// TwinCAT 3 PLC project Sample01
// ProgramVersion: 3.1.4023.0
// libraries:
//   Tc2_Standard, * (Beckhoff Automation GmbH)
//   Tc2_System, * (Beckhoff Automation GmbH)
//   Tc3_Module, * (Beckhoff Automation GmbH)
// project tree:
//   DUTs/ E_SortedOrder.TcDUT, ST_SequenceItem.TcDUT
//   / PlcTask.TcTTO
//   POUs/ Class Diagram.TcCD (not stored), FB_SequenceManager.TcPOU, MAIN.TcPOU
// real-time tasks:
//   TASK PlcTask: cycle T#10ms, priority 20, ADS port 350

CONFIGURATION Sample01
    RESOURCE PLC ON TwinCAT3
        TASK PlcTask(INTERVAL := T#10ms, PRIORITY := 20);
        PROGRAM MAIN WITH PlcTask : MAIN;
    END_RESOURCE
END_CONFIGURATION

// ---- DUTs/E_SortedOrder.TcDUT
{attribute 'qualified_only'}
{attribute 'strict'}
TYPE E_SortedOrder :
(
	Id,
	Value
);
END_TYPE

// ---- DUTs/ST_SequenceItem.TcDUT
TYPE ST_SequenceItem :
STRUCT
	nId			: UINT;
	nValue		: USINT(0..100);
	nDuration	: UINT; 
END_STRUCT
END_TYPE

// ---- POUs/MAIN.TcPOU
PROGRAM MAIN
VAR
	fbPlayList		: FB_SequenceManager;
	nTest			: INT;
END_VAR

IF (nTest = 1) THEN
	fbPlayList.Sort(E_SortedOrder.Id);
	nTest := 0;
ELSIF (nTest = 2) THEN
	fbPlayList.Sort(E_SortedOrder.Value);
	nTest := 0;
END_IF

END_PROGRAM

// ---- POUs/FB_SequenceManager.TcPOU
FUNCTION_BLOCK PUBLIC FB_SequenceManager
VAR_INPUT
END_VAR
VAR_OUTPUT
END_VAR
VAR
	// backing variable
	_aSequence	: ARRAY [1..5] OF ST_SequenceItem := [(nId := 1, nValue := 50, nDuration := 20),
													  (nId := 2, nValue := 10, nDuration := 30),
													  (nId := 3, nValue := 23, nDuration := 10),
													  (nId := 4, nValue := 65, nDuration := 200),
													  (nId := 5, nValue := 45, nDuration := 75)];
END_VAR

{attribute 'monitoring' := 'variable'}
PROPERTY PUBLIC aSequence : ARRAY [1..5] OF ST_SequenceItem
GET
aSequence := _aSequence;
END_GET
SET // PROTECTED
_aSequence := aSequence;
END_SET
END_PROPERTY

METHOD PUBLIC Sort
VAR_INPUT
	eSortedOrder		: E_SortedOrder;
END_VAR
VAR
	stLeft, stRight		: ST_SequenceItem;
	nMax, nIndex		: DINT;
	bSwapped			: BOOL;
END_VAR
CASE eSortedOrder OF
	E_SortedOrder.Id:
		REPEAT
			bSwapped := FALSE;
			FOR nIndex := 1 TO 4 DO
				stLeft := THIS^._aSequence[nIndex];
				stRight := THIS^._aSequence[nIndex + 1];
				IF (stLeft.nId > stRight.nId) THEN
					THIS^._aSequence[nIndex + 1] := stLeft;
					THIS^._aSequence[nIndex] := stRight;
					bSwapped := TRUE;
				END_IF
			END_FOR
		UNTIL
			bSwapped = FALSE
		END_REPEAT;

	E_SortedOrder.Value:
		REPEAT
			bSwapped := FALSE;
			FOR nIndex := 1 TO 4 DO
				stLeft := THIS^._aSequence[nIndex];
				stRight := THIS^._aSequence[nIndex + 1];
				IF (stLeft.nValue > stRight.nValue) THEN
					THIS^._aSequence[nIndex + 1] := stLeft;
					THIS^._aSequence[nIndex] := stRight;
					bSwapped := TRUE;
				END_IF
			END_FOR
		UNTIL
			bSwapped = FALSE
		END_REPEAT;
END_CASE
END_METHOD

END_FUNCTION_BLOCK
